ABB RAPID module: ConfigUser.mod

MODULE ConfigUser
!*************************************
!* Module which contains data global *
!*      to all T_Rob1 modules        *
!*************************************
!# -----------------------
!# ------ Tooldata
!# -----------------------
PERS tooldata t_Grp1:=[TRUE, [[26.5774,98.0613,502.695],[0.608761,0,0,-0.793353]], [311.4, [-15.6,-0.4,261.4],[1,0,0,0], 130.469,118.237,123.004]];
PERS tooldata t_Grp1_Roll:=[True, [[-75.715912,494.028526,713.989449],[0.608668,0.000878,0.000753,-0.793424]], [317.6, [-11.9,0.9,267.3],[1,0,0,0], 87.053,155.869,134.128]];

!# -----------------------
!# ------ Wobjdata
!# -----------------------
PERS wobjdata wobj_65fx02:=[False,True,"",[[-1620.001874,-2435.035666,-422.236299],[0.653281,-0.270598,-0.270598,-0.653282]],[[0,0,0],[1,0,0,0]]];
PERS wobjdata wobj_65fx01:=[False,True,"",[[602.999931,2050.006628,-515.000122],[0,0,0,1]],[[0,0,0],[1,0,0,0]]];
PERS wobjdata wobj_65fx01_best_fit:=[FALSE,TRUE,"",[[603,2050.01,-515],[0,0,0,1]],[[0.067,1.318,1.054],[0.999999,0.000898756,8.81684E-05,0.00100349]]];
PERS wobjdata wobj_calibration:=[False,True,"",[[494.999926,-2309.463648,-960.934326],[0.653281,-0.270598,0.270598,0.653281]],[[0,0,0],[1,0,0,0]]];

!# -----------------------
!# ------ Loaddata
!# -----------------------
PERS loaddata ld_Bonnet_f56:=[21.2,[106,-5.7,-96.4],[1,0,0,0],1.6,12.1,6.1];
PERS tooldata t_BCF_F55:=[TRUE,[[26.5774,98.0613,502.695],[0.00656,-0.61393,0.78928,0.00936]],[311.4,[-15.6,-0.4,261.4],[1,0,0,0],130.469,118.237,123.004]];

!# -----------------------
!# ------ Numdata
!# -----------------------

!# -----------------------
!# ------ Booldata
!# -----------------------

!# -----------------------
!# ------ Speeddata
!# -----------------------

!# -----------------------
!# ------ Jointdata
!# -----------------------

!# -----------------------
!# ------ Stringdata
!# -----------------------
PERS string RecordTime01;
PERS string RecordTime02;
PERS string RecordTime03;
PERS string RecordTime04;


!# -----------------------
!# ------ Robtargetdata
!# -----------------------

ENDMODULE
